FUNCTION_BLOCK PUBLIC FB_ItalianPizzaSalami EXTENDS FB_ItalianPizzaMargherita
VAR_INPUT
END_VAR
VAR_OUTPUT
END_VAR
VAR
	bSalami		: BOOL := TRUE;
END_VAR

PROPERTY PUBLIC bHasSalami : BOOL
GET
bHasSalami := this^.bSalami;
END_GET
SET
this^.bSalami := bHasSalami;
END_SET
END_PROPERTY

METHOD PUBLIC GetPrice : LREAL
GetPrice := SUPER^.GetPrice();
IF (THIS^.bSalami) THEN
	GetPrice := GetPrice + 1.4;
END_IF
END_METHOD

END_FUNCTION_BLOCK

(* stored: Version 1.1.0.1, ProductVersion 3.1.4022.12
   POU FB_ItalianPizzaSalami: Id {f9e0a7fb-5319-4a7b-a1d3-599810cef0e9}, SpecialFunc None
   Property bHasSalami: Id {22bb5d10-0476-4a6f-854e-2e8862b0178e}
   Get Get: Id {6ea39efb-5e8c-4fbf-9db6-206cb00c8b2a}
   Set Set: Id {2ab1f08e-af77-4aad-89fa-85ecc19e2652}
   Method GetPrice: Id {61451c2b-8fe9-41cb-9877-0912f6cd0e4f} *)
